Yaskawa INFORM job: HANDSHAK.JBI

/JOB
//NAME HANDSHAK
//POS
///NPOS 0,0,0,0,0,0
//INST
///DATE 2015/04/28 15:16
///ATTR SC,RW,MC
///LVARS 5,5,5,5,0,0,0,0
NOP
GETARG LB000 IARG#(1)
DOUT OG#(68) LB[0]
END
